// TIA Portal V20 export
TYPE "zp_CITIEoC"
// stored: Access Published, Namespace CITI_Logic
   STRUCT
      PUN_Ready : Bool;
      FTQ_DataReady : Bool;
      Energy_Conservation_Enable : Bool;
      Buffer_Bypassed : Bool;
      Bypassed : Bool;
      Safety_Checksum_OK : Bool;
      Spare_7 : Bool;
      Spare_8 : Bool;
      Spare_SINT : SInt;
      Spare_INT : Int;
      PUN_Data : String[20];   // PUN Data
      FTQ_PUN_Data : String[20];
      PUN_GM_Part_Num : String[8];
      PUN_Optional_Data : String[12];
      Part_Type : String[12];
      Reject_Message : String[100];
      AOI_Revision : Int;
      Good_Count : Int;
      Reject_Count : Int;
      Buffer_Count : Int;
      LastLoadTime : Int;
      LastUnloadTIme : Int;
      Part_Type_Message : Int;
      Bypassed_Pallet_Count : Int;
      Filter_Current_Temp : Int;
      Filter_NumQuantity_1 : Int;
      Filter_NumQuantity_2 : Int;
      Filter_NumQuantity_3 : Int;
      Spare_INT_2 : Int;
      Rated_Cycle_Time : DInt;
      Last_Cycle_Time : DInt;
      LastProcessingTime : DInt;
      Reject_Code : DInt;
   END_STRUCT;
END_TYPE
